TYPE RxData :
STRUCT
  Command : UINT;         // Echoed command code
  Data : ARRAY[0..5] OF BYTE; // 6 bytes for response data
END_STRUCT
END_TYPE

(* stored: Version 1.1.0.1, ProductVersion 3.1.4024.13
   DUT RxData: Id {e41e376b-7ae2-467e-a614-ddb07fab5b6b} *)
